TYPE T_NOTT_CRYO_WARMUP_CTRL :
STRUCT
	

END_STRUCT
END_TYPE

(* stored: Version 1.1.0.1, ProductVersion 3.1.4026.18
   DUT T_NOTT_CRYO_WARMUP_CTRL: Id {1bd6dc4c-40ac-401c-bf2b-1f228abdc631} *)
